INTERFACE IWaitVariableValueActivity EXTENDS IActivity

METHOD Configure
VAR_INPUT
	monitoredVariableName : STRING;
	referenceValue : ANY; 
END_VAR
END_METHOD

{attribute 'monitoring' := 'call'}
PROPERTY MonitoredVariableName : STRING
GET
END_GET
END_PROPERTY

{attribute 'monitoring' := 'call'}
PROPERTY ReferenceValue : __SYSTEM.AnyType
GET
END_GET
END_PROPERTY

END_INTERFACE

(* stored: Version 1.1.0.1
   Itf IWaitVariableValueActivity: Id {4709ad70-25c3-4af9-87d2-a6abbd569ae5}
   Method Configure: Id {81bca520-5ab8-463c-aa20-d6acbb1890b1}
   Property MonitoredVariableName: Id {ff4d8127-2610-427d-98b2-05f651f24b0a}
   Get Get: Id {5829b1fb-5931-4f2d-a0f0-282256597065}
   Property ReferenceValue: Id {617dba7f-5920-42d0-9d1e-c0ec1975c92a}
   Get Get: Id {b3a72245-5245-4e15-be7b-53b88c5316a9} *)
